// SIMATIC S7-200 project (STEP 7-Micro/WIN), CPU 224 REL 01.11

SYMBOL_TABLE USER1
ONN              I0.0
DEN1             Q0.0
DEN2             Q0.1
END_SYMBOL_TABLE

ORGANIZATION_BLOCK MAIN:OB1
TITLE=PROGRAM COMMENTS
BEGIN
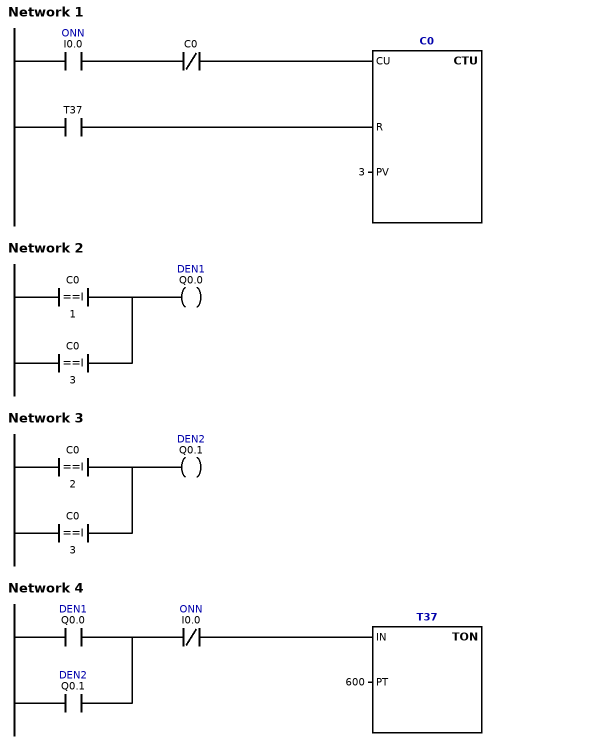
Network 1
LD     ONN:I0.0
AN     C0
LD     T37
CTU    C0, 3
Network 2
LDW=   C0, 1
OW=    C0, 3
=      DEN1:Q0.0
Network 3
LDW=   C0, 2
OW=    C0, 3
=      DEN2:Q0.1
Network 4
LD     DEN1:Q0.0
O      DEN2:Q0.1
AN     ONN:I0.0
TON    T37, 600
END_ORGANIZATION_BLOCK
